{attribute 'linkalways'} 
{attribute 'no_explicit_call' := 'This FB is a CLASS and must be accessed using methods or properties'}
{attribute 'enable_dynamic_creation'}
FUNCTION_BLOCK _Array0to3OfDINT EXTENDS ArrayDatatypeBase
VAR CONSTANT
	lBound : DINT := 0;
	uBound : DINT := 3;
END_VAR
VAR
	localData : ARRAY [lBound..uBound] OF DINT;
	activeData : REFERENCE TO ARRAY [lBound..uBound] OF DINT REF= localData;
	elements : ARRAY [lBound..uBound] OF _DINT(0);
	baseType : _DINT(0);
END_VAR

PROPERTY PUBLIC Address : PVOID
GET
Address := ADR(activeData);
END_GET
END_PROPERTY

PROPERTY PUBLIC BaseDatatype : I_Datatype
GET
BaseDatatype := baseType;
END_GET
END_PROPERTY

METHOD PUBLIC ClearReference
VAR_INPUT
END_VAR
activeData REF= localData;
SetElementReference();
END_METHOD

METHOD PUBLIC Clone : I_Datatype
VAR
    pClone : POINTER TO _Array0to3OfDINT;
END_VAR
pClone := __NEW(_Array0to3OfDINT());
pClone^.Value := Value;
Clone := pClone^;
END_METHOD

METHOD FB_init : BOOL
VAR_INPUT
	bInitRetains : BOOL; // if TRUE, the retain variables are initialized (warm start / cold start)
	bInCopyCode : BOOL;  // if TRUE, the instance afterwards gets moved into the copy code (online change)
END_VAR
SetElementReference();
END_METHOD

METHOD PUBLIC GetElementAsDatatypeByIndex : I_Datatype
VAR_INPUT
	Index : DINT;
END_VAR
GetElementAsDatatypeByIndex := elements[Index];
END_METHOD

METHOD PUBLIC GetElementByIndex : REFERENCE TO _DINT;
VAR_INPUT
	Index : DINT;
END_VAR
GetElementByIndex REF= elements[Index];
END_METHOD

PROPERTY PUBLIC LowerBound : DINT
GET
LowerBound := lBound;
END_GET
END_PROPERTY

METHOD PUBLIC MakeReferenceTo
VAR_INPUT
	ReferenceTarget : REFERENCE TO ARRAY [lBound..uBound] OF DINT;
END_VAR
activeData REF= ReferenceTarget;
SetElementReference();
END_METHOD

METHOD PROTECTED OnSerializeArrayValues
VAR_INPUT
	Serializer : I_Serializer;
END_VAR
VAR
	i : DINT;
END_VAR
FOR i := lBound TO uBound DO
	elements[i].SerializeWith(Serializer);
END_FOR
END_METHOD

METHOD PROTECTED SetElementReference
VAR_INPUT
END_VAR
VAR
	i : DINT;
END_VAR
FOR i := lBound TO uBound DO
	elements[i].MakeReferenceTo(activeData[i]);
END_FOR
END_METHOD

PROPERTY PUBLIC Size : UDINT
GET
Size := SIZEOF(activeData);
END_GET
END_PROPERTY

METHOD PROTECTED TryDeserializeArrayValues : BOOL
VAR_INPUT
	Deserializer : I_Deserializer;
	Feedback : I_DeserializerFeedback;
END_VAR
VAR
	enumerator : I_DeserializerArrayForwardEnumerator;
	i : DINT;
END_VAR
enumerator := Deserializer.GetArrayEnumerator();
i := lBound;

WHILE enumerator.MoveNext() AND i <= uBound DO
	
	IF NOT elements[i].TryDeserializeFrom(enumerator.Current, Feedback) THEN
		EXIT;
	END_IF
	i := i + 1;

END_WHILE
enumerator.Dispose();
END_METHOD

METHOD TryMakeReferenceTo : BOOL
VAR_INPUT
	Target : I_Datatype;
END_VAR
VAR
	targetAsArray : I_ArrayDatatype;
	pTargetData : POINTER TO ARRAY [lBound..uBound] OF DINT;
END_VAR
IF NOT Target.TryResolveAsArrayDatatype(targetAsArray) THEN
	RETURN;
END_IF

IF NOT (targetAsArray.Identifier = Identifier) THEN
	RETURN;
END_IF

pTargetData := Target.Address;
activeData REF= pTargetData^;
SetElementReference();
TryMakeReferenceTo := TRUE;
END_METHOD

PROPERTY PUBLIC UpperBound : DINT
GET
UpperBound := ubound;
END_GET
END_PROPERTY

PROPERTY PUBLIC Value : REFERENCE TO ARRAY [lBound..uBound] OF DINT;
GET
Value ref= activeData;
END_GET
END_PROPERTY

END_FUNCTION_BLOCK

(* stored: Version 1.1.0.1, ProductVersion 3.1.4024.13
   POU _Array0to3OfDINT: Id {64a20a04-94cb-03b2-2a14-f0500ee8ce46}, SpecialFunc None
   Folder Core: Id {f8acbd12-a5cc-0525-3c81-8f8b9a4b68b7}
   Folder Constructor: Id {8dee56db-0912-08b0-0010-aa9e6f7408b0}
   Folder Protected: Id {53bf86b5-7b2b-020e-3377-ac68d0836d98}
   Folder Customize: Id {7086d3e1-f8ff-01a0-121e-4531e80989d8}
   Property Address: Id {e0adc1bb-5d61-0748-0c2c-bda44e41f9c5}
   Get Get: Id {6ca9fd3b-231c-0e17-27ea-b9feaaf8053c}
   Property BaseDatatype: Id {01480af5-5238-080a-1c33-a3110b821447}
   Get Get: Id {69262443-2fb1-082d-255e-58376af08353}
   Method ClearReference: Id {fc7f4b3b-513f-0062-38b7-43c9edb7f63c}
   Method Clone: Id {3eeb34a1-f8f1-07a3-1aaa-bf7bd3a1726f}
   Method FB_init: Id {7e14dd9f-8e91-0087-2a48-8fc81f3f7d52}
   Method GetElementAsDatatypeByIndex: Id {16349904-1747-03ed-03e1-1490d4734f4b}
   Method GetElementByIndex: Id {bf6eef4a-9413-0c51-0cc3-dfd66d34838c}
   Property LowerBound: Id {e1cf66fa-3ebf-0251-3a99-0e6e8a35b35f}
   Get Get: Id {5a5d48cf-32e8-08ed-1ff3-37272d0fb2e8}
   Method MakeReferenceTo: Id {0883f8ed-e936-019f-02b6-3c5ede4e5518}
   Method OnSerializeArrayValues: Id {bb17ba47-a2bc-088c-1af1-66b7dd1e0ec9}
   Method SetElementReference: Id {3b0e2188-b3b1-001a-15fb-4699790787d1}
   Property Size: Id {39ab5f20-e922-0dfc-0a3d-1728d70081fd}
   Get Get: Id {e4ad3711-2eab-003e-35c2-a13cac7df1da}
   Method TryDeserializeArrayValues: Id {92d7b224-d09a-0c1f-2c8d-05f1fe82d3e4}
   Method TryMakeReferenceTo: Id {64093090-93ca-0771-0ae4-b7f39e4c39d5}
   Property UpperBound: Id {3befda24-42ec-07d2-1205-b0dd868de349}
   Get Get: Id {ff098539-cdec-0361-21b6-b6ed961794ca}
   Property Value: Id {69a4f9fe-17e0-0f0c-3644-8e604e6734fe}
   Get Get: Id {e3e86e7b-b012-08e6-3328-6f4e06c3e183} *)
